// Mitsubishi GX Works2 project: m06   PLC: Q02/Q02H

PROGRAM MAIN
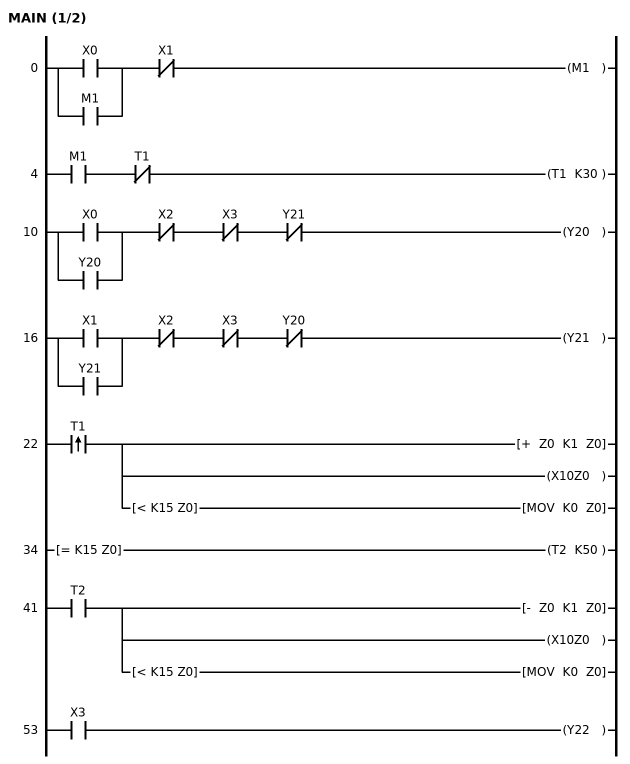
0     LD      X0
      OR      M1
      ANI     X1
      OUT     M1
4     LD      M1
      ANI     T1
      OUT     T1 K30
10    LD      X0
      OR      Y20
      ANI     X2
      ANI     X3
      ANI     Y21
      OUT     Y20
16    LD      X1
      OR      Y21
      ANI     X2
      ANI     X3
      ANI     Y20
      OUT     Y21
22    LDP     T1
      +       Z0 K1 Z0
      OUT     X10Z0
      AND<    K15 Z0
      MOV     K0 Z0
34    LD=     K15 Z0
      OUT     T2 K50
41    LD      T2
      -       Z0 K1 Z0
      OUT     X10Z0
      AND<    K15 Z0
      MOV     K0 Z0
53    LD      X3
      OUT     Y22
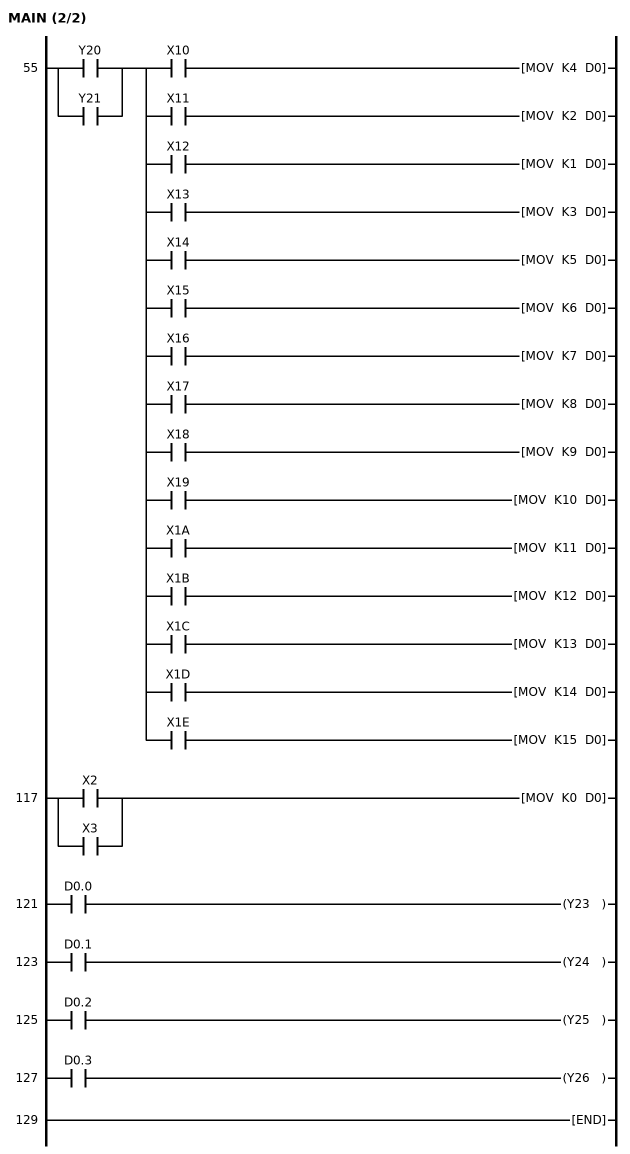
55    LD      Y20
      OR      Y21
      MPS
      AND     X10
      MOV     K4 D0
      MRD
      AND     X11
      MOV     K2 D0
      MRD
      AND     X12
      MOV     K1 D0
      MRD
      AND     X13
      MOV     K3 D0
      MRD
      AND     X14
      MOV     K5 D0
      MRD
      AND     X15
      MOV     K6 D0
      MRD
      AND     X16
      MOV     K7 D0
      MRD
      AND     X17
      MOV     K8 D0
      MRD
      AND     X18
      MOV     K9 D0
      MRD
      AND     X19
      MOV     K10 D0
      MRD
      AND     X1A
      MOV     K11 D0
      MRD
      AND     X1B
      MOV     K12 D0
      MRD
      AND     X1C
      MOV     K13 D0
      MRD
      AND     X1D
      MOV     K14 D0
      MPP
      AND     X1E
      MOV     K15 D0
117   LD      X2
      OR      X3
      MOV     K0 D0
121   LD      D0.0
      OUT     Y23
123   LD      D0.1
      OUT     Y24
125   LD      D0.2
      OUT     Y25
127   LD      D0.3
      OUT     Y26
129   END
END_PROGRAM
